RoboDK station: path.rdk

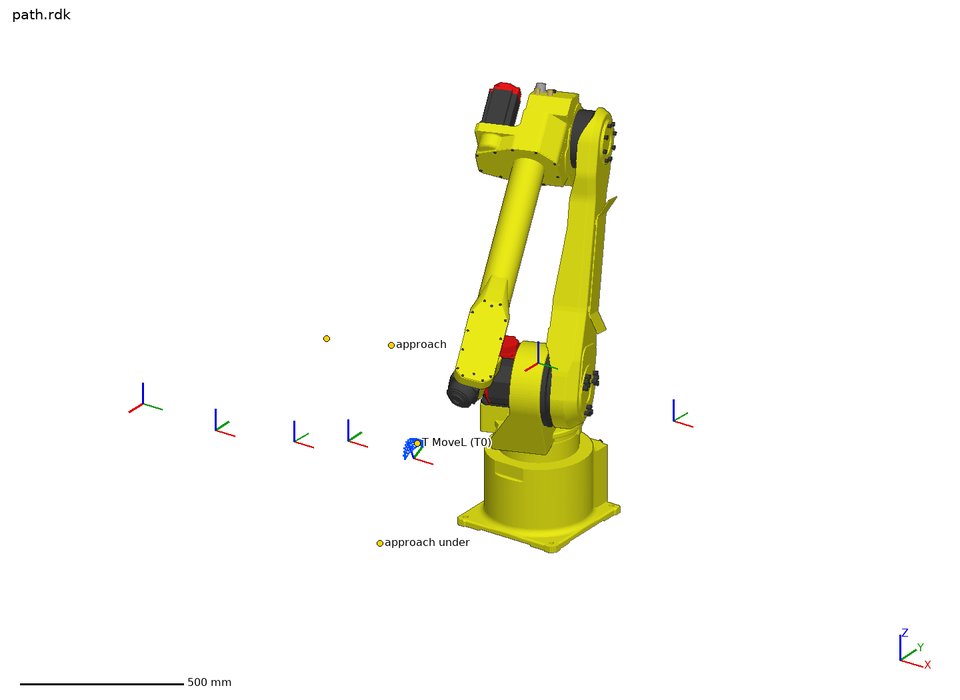
[picture v0: the station drawn from its stored meshes, robots at their saved joint values, targets as dots, program paths as lines]
Station path (saved by RoboDK 5.0.0). Poses are relative to the parent item; angles as X-Y-Z fixed-axis rotations.
  - frame data_frame at (0, 0, 0) mm
    - target approach (Cartesian target) at (94, 380, 204.2) mm, rotated rx -180 ry 0 rz 0 deg; joints [10.247, -49.52, -8.659, -50.211, 13.385, 139.433] of Fanuc ARC Mate 120iB/10L
    - target approach_vert (Cartesian target) at (0, 170, 284.2) mm, rotated rx -90 ry 0 rz 180 deg; joints [0, 2.156, 3.881, -180, 93.881, 90] of Fanuc ARC Mate 120iB/10L
    - target approach under (Cartesian target) at (94, 320, -445.8) mm; joints [3.897, 48.417, -53.03, 175.127, 126.871, 267.072] of Fanuc ARC Mate 120iB/10L
    - target approach_vert_180 (Cartesian target) at (0, 170, 284.2) mm, rotated rx -90 ry 0 rz 0 deg; joints [0, 2.156, 3.881, -180, 93.881, -90] of Fanuc ARC Mate 120iB/10L
    - frame data_frame_sphere at (270, 250, -80) mm, rotated rx 25 ry 0 rz 0 deg
      - object path at (0, 0, 0) mm, geometry from ible
      - target T MoveL (T0) (Cartesian target) at (-12.84, 46.05, 14.64) mm, rotated rx 112.92 ry -41.25 rz 0 deg; joints [16.302, 22.375, -63.434, -8.779, 128.992, 144.295] of Fanuc ARC Mate 120iB/10L
    - frame data_frame_zcyl at (-610, 450, -310) mm
    - frame data_frame_ycyl at (890, 750, 20) mm
    - frame data_frame_xcyl at (130, 100, 0) mm
    - frame data_frame_delta at (-1050, 690, -440) mm, rotated rx 0 ry 0 rz -90 deg
  - frame Fanuc ARC Mate 120iB/10L Base at (0, 1300, -250) mm, rotated rx 0 ry 0 rz -90 deg
    - robot Fanuc ARC Mate 120iB/10L: 6 axes, payload 10 kg, reach 1885 mm, repeatability 0.1 mm, weight 225 kg
        modified DH rows (alpha deg, a mm, theta deg, d mm): 0, 0, 0, 525; -90, 150, -90, 0; 0, 770, 0, 0; -90, 100, 0, 960; 90, 0, 0, 0; -90, 0, 0, 100
        base shift (0, 0, -525) mm
        joint limits [-170, -80, -170, -200, -140, -2160] to [170, 170, 250, 200, 140, 2160]; home [0, 0, 0, 0, 0, 0]; saved at [20.227, -18.261, -31.301, 104.445, -18.879, 20.92]
      - tool Tool 1, TCP at (0, 0, 300) mm, rotated rx 90 ry 0 rz 0 deg
      - tool Tool Normal, TCP at (0, 0, 200) mm
      - tool Tool 3, TCP at (0, 0, 300) mm, rotated rx -90 ry 0 rz 0 deg
      - tool Tool OD Orient, TCP at (0, 0, 300) mm, rotated rx 0 ry 90 rz -90 deg
      - tool Tool Sphere, TCP at (0, 0, 200) mm, rotated rx 0 ry 0 rz 45 deg
  - program AutoProgram (201 instructions, listed below)
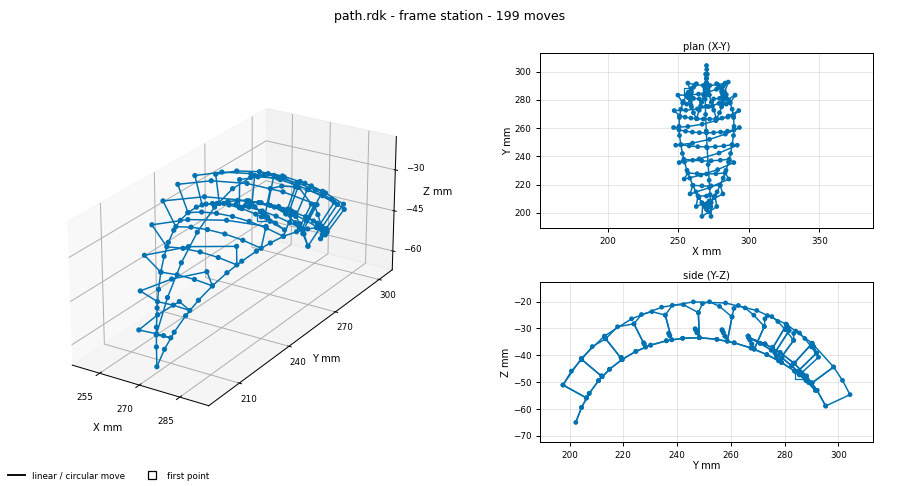
[picture p0: tool path of path.rdk in frame station, 199 of 199 moves have a stored position in this frame; points joined in program order, loops and branches not executed]

--- program AutoProgram (robot Fanuc ARC Mate 120iB/10L) ---
  Set Ref.: data_frame_sphere
  Set Tool: Tool Sphere
  *MoveL (T0) -> target T MoveL (T0)
  MoveL (T1) to (-11.94, 46.05, 15.38) mm, rotated rx 112.92 ry -37.81 rz 0 deg; joints [16.302, 22.375, -63.434, -8.779, 128.992, 144.295]
  MoveL (T2) to (-10.99, 46.05, 16.07) mm, rotated rx 112.92 ry -34.38 rz 0 deg; joints [16.302, 22.375, -63.434, -8.779, 128.992, 144.295]
  MoveL (T3) to (-13.19, 55.26, 19.28) mm, rotated rx 112.92 ry -34.38 rz 0 deg; joints [16.302, 22.375, -63.434, -8.779, 128.992, 144.295]
  MoveL (T4) to (-8.01, 55.26, 21.95) mm, rotated rx 112.92 ry -20.05 rz 0 deg; joints [16.302, 22.375, -63.434, -8.779, 128.992, 144.295]
  MoveL (T5) to (-2.33, 55.26, 23.25) mm, rotated rx 112.92 ry -5.73 rz 0 deg; joints [16.302, 22.375, -63.434, -8.779, 128.992, 144.295]
  MoveL (T6) to (-1.94, 46.05, 19.37) mm, rotated rx 112.92 ry -5.73 rz 0 deg; joints [16.302, 22.375, -63.434, -8.779, 128.992, 144.295]
  MoveL (T7) to (0, 46.05, 19.47) mm, rotated rx 112.92 ry 0 rz 0 deg; joints [16.302, 22.375, -63.434, -8.779, 128.992, 144.295]
  MoveL (T8) to (1.94, 46.05, 19.37) mm, rotated rx 112.92 ry 5.73 rz 0 deg; joints [16.302, 22.375, -63.434, -8.779, 128.992, 144.295]
  MoveL (T9) to (2.33, 55.26, 23.25) mm, rotated rx 112.92 ry 5.73 rz 0 deg; joints [16.302, 22.375, -63.434, -8.779, 128.992, 144.295]
  MoveL (T10) to (8.01, 55.26, 21.95) mm, rotated rx 112.92 ry 20.05 rz 0 deg; joints [16.302, 22.375, -63.434, -8.779, 128.992, 144.295]
  MoveL (T11) to (13.19, 55.26, 19.28) mm, rotated rx 112.92 ry 34.38 rz 0 deg; joints [16.302, 22.375, -63.434, -8.779, 128.992, 144.295]
  MoveL (T12) to (10.99, 46.05, 16.07) mm, rotated rx 112.92 ry 34.38 rz 0 deg; joints [16.302, 22.375, -63.434, -8.779, 128.992, 144.295]
  MoveL (T13) to (11.94, 46.05, 15.38) mm, rotated rx 112.92 ry 37.81 rz 0 deg; joints [16.302, 22.375, -63.434, -8.779, 128.992, 144.295]
  MoveL (T14) to (12.84, 46.05, 14.64) mm, rotated rx 112.92 ry 41.25 rz 0 deg; joints [16.302, 22.375, -63.434, -8.779, 128.992, 144.295]
  MoveL (T15) to (15.41, 55.26, 17.57) mm, rotated rx 112.92 ry 41.25 rz 0 deg; joints [16.302, 22.375, -63.434, -8.779, 128.992, 144.295]
  MoveL (T16) to (11.93, 54.45, 22.19) mm, rotated rx 114.83 ry 28.27 rz 0 deg; joints [16.302, 22.375, -63.434, -8.779, 128.992, 144.295]
  MoveL (T17) to (7.11, 53.58, 26.04) mm, rotated rx 116.74 ry 15.28 rz 0 deg; joints [16.302, 22.375, -63.434, -8.779, 128.992, 144.295]
  MoveL (T18) to (1.15, 52.66, 28.74) mm, rotated rx 118.65 ry 2.29 rz 0 deg; joints [16.302, 22.375, -63.434, -8.779, 128.992, 144.295]
  MoveL (T19) to (-5.66, 51.67, 29.97) mm, rotated rx 120.56 ry -10.7 rz 0 deg; joints [16.302, 22.375, -63.434, -8.779, 128.992, 144.295]
  MoveL (T20) to (-12.94, 50.62, 29.5) mm, rotated rx 122.47 ry -23.68 rz 0 deg; joints [16.302, 22.375, -63.434, -8.779, 128.992, 144.295]
  MoveL (T21) to (-20.23, 49.52, 27.17) mm, rotated rx 124.38 ry -36.67 rz 0 deg; joints [16.302, 22.375, -63.434, -8.779, 128.992, 144.295]
  MoveL (T22) to (-16.86, 41.27, 22.64) mm, rotated rx 124.38 ry -36.67 rz 0 deg; joints [16.302, 22.375, -63.434, -8.779, 128.992, 144.295]
  MoveL (T23) to (-14.03, 41.27, 24.5) mm, rotated rx 124.38 ry -29.79 rz 0 deg; joints [16.302, 22.375, -63.434, -8.779, 128.992, 144.295]
  MoveL (T24) to (-10.99, 41.27, 26) mm, rotated rx 124.38 ry -22.92 rz 0 deg; joints [16.302, 22.375, -63.434, -8.779, 128.992, 144.295]
  MoveL (T25) to (-13.19, 49.52, 31.2) mm, rotated rx 124.38 ry -22.92 rz 0 deg; joints [16.302, 22.375, -63.434, -8.779, 128.992, 144.295]
  MoveL (T26) to (-9.2, 49.52, 32.61) mm, rotated rx 124.38 ry -15.76 rz 0 deg; joints [16.302, 22.375, -63.434, -8.779, 128.992, 144.295]
  MoveL (T27) to (-5.06, 49.52, 33.5) mm, rotated rx 124.38 ry -8.59 rz 0 deg; joints [16.302, 22.375, -63.434, -8.779, 128.992, 144.295]
  MoveL (T28) to (-4.22, 41.27, 27.91) mm, rotated rx 124.38 ry -8.59 rz 0 deg; joints [16.302, 22.375, -63.434, -8.779, 128.992, 144.295]
  MoveL (T29) to (0, 41.27, 28.23) mm, rotated rx 124.38 ry 0 rz 0 deg; joints [16.302, 22.375, -63.434, -8.779, 128.992, 144.295]
  MoveL (T30) to (4.22, 41.27, 27.91) mm, rotated rx 124.38 ry 8.59 rz 0 deg; joints [16.302, 22.375, -63.434, -8.779, 128.992, 144.295]
  MoveL (T31) to (5.06, 49.52, 33.5) mm, rotated rx 124.38 ry 8.59 rz 0 deg; joints [16.302, 22.375, -63.434, -8.779, 128.992, 144.295]
  MoveL (T32) to (9.2, 49.52, 32.61) mm, rotated rx 124.38 ry 15.76 rz 0 deg; joints [16.302, 22.375, -63.434, -8.779, 128.992, 144.295]
  MoveL (T33) to (13.19, 49.52, 31.2) mm, rotated rx 124.38 ry 22.92 rz 0 deg; joints [16.302, 22.375, -63.434, -8.779, 128.992, 144.295]
  MoveL (T34) to (10.99, 41.27, 26) mm, rotated rx 124.38 ry 22.92 rz 0 deg; joints [16.302, 22.375, -63.434, -8.779, 128.992, 144.295]
  MoveL (T35) to (14.03, 41.27, 24.5) mm, rotated rx 124.38 ry 29.79 rz 0 deg; joints [16.302, 22.375, -63.434, -8.779, 128.992, 144.295]
  MoveL (T36) to (16.86, 41.27, 22.64) mm, rotated rx 124.38 ry 36.67 rz 0 deg; joints [16.302, 22.375, -63.434, -8.779, 128.992, 144.295]
  MoveL (T37) to (20.23, 49.52, 27.17) mm, rotated rx 124.38 ry 36.67 rz 0 deg; joints [16.302, 22.375, -63.434, -8.779, 128.992, 144.295]
  MoveL (T38) to (15.12, 48.36, 32.13) mm, rotated rx 126.29 ry 25.21 rz 0 deg; joints [16.302, 22.375, -63.434, -8.779, 128.992, 144.295]
  MoveL (T39) to (8.82, 47.15, 36.04) mm, rotated rx 128.2 ry 13.75 rz 0 deg; joints [16.302, 22.375, -63.434, -8.779, 128.992, 144.295]
  MoveL (T40) to (1.55, 45.89, 38.62) mm, rotated rx 130.11 ry 2.29 rz 0 deg; joints [16.302, 22.375, -63.434, -8.779, 128.992, 144.295]
  MoveL (T41) to (-6.4, 44.58, 39.65) mm, rotated rx 132.02 ry -9.17 rz 0 deg; joints [16.302, 22.375, -63.434, -8.779, 128.992, 144.295]
  MoveL (T42) to (-14.66, 43.21, 38.96) mm, rotated rx 133.93 ry -20.63 rz 0 deg; joints [16.302, 22.375, -63.434, -8.779, 128.992, 144.295]
  MoveL (T43) to (-22.86, 41.8, 36.47) mm, rotated rx 135.84 ry -32.09 rz 0 deg; joints [16.302, 22.375, -63.434, -8.779, 128.992, 144.295]
  MoveL (T44) to (-19.05, 34.84, 30.39) mm, rotated rx 135.84 ry -32.09 rz 0 deg; joints [16.302, 22.375, -63.434, -8.779, 128.992, 144.295]
  MoveL (T45) to (-15.13, 34.84, 32.52) mm, rotated rx 135.84 ry -24.96 rz 0 deg; joints [16.302, 22.375, -63.434, -8.779, 128.992, 144.295]
  MoveL (T46) to (-10.98, 34.84, 34.15) mm, rotated rx 135.84 ry -17.83 rz 0 deg; joints [16.302, 22.375, -63.434, -8.779, 128.992, 144.295]
  MoveL (T47) to (-6.66, 34.84, 35.24) mm, rotated rx 135.84 ry -10.7 rz 0 deg; joints [16.302, 22.375, -63.434, -8.779, 128.992, 144.295]
  MoveL (T48) to (-2.23, 34.84, 35.8) mm, rotated rx 135.84 ry -3.56 rz 0 deg; joints [16.302, 22.375, -63.434, -8.779, 128.992, 144.295]
  MoveL (T49) to (2.23, 34.84, 35.8) mm, rotated rx 135.84 ry 3.56 rz 0 deg; joints [16.302, 22.375, -63.434, -8.779, 128.992, 144.295]
  MoveL (T50) to (6.66, 34.84, 35.24) mm, rotated rx 135.84 ry 10.7 rz 0 deg; joints [16.302, 22.375, -63.434, -8.779, 128.992, 144.295]
  MoveL (T51) to (10.98, 34.84, 34.15) mm, rotated rx 135.84 ry 17.83 rz 0 deg; joints [16.302, 22.375, -63.434, -8.779, 128.992, 144.295]
  MoveL (T52) to (15.13, 34.84, 32.52) mm, rotated rx 135.84 ry 24.96 rz 0 deg; joints [16.302, 22.375, -63.434, -8.779, 128.992, 144.295]
  MoveL (T53) to (19.05, 34.84, 30.39) mm, rotated rx 135.84 ry 32.09 rz 0 deg; joints [16.302, 22.375, -63.434, -8.779, 128.992, 144.295]
  MoveL (T54) to (22.86, 41.8, 36.47) mm, rotated rx 135.84 ry 32.09 rz 0 deg; joints [16.302, 22.375, -63.434, -8.779, 128.992, 144.295]
  MoveL (T55) to (15.4, 40.05, 41.94) mm, rotated rx 138.13 ry 20.17 rz 0 deg; joints [16.302, 22.375, -63.434, -8.779, 128.992, 144.295]
  MoveL (T56) to (6.64, 38.23, 45.77) mm, rotated rx 140.42 ry 8.25 rz 0 deg; joints [16.302, 22.375, -63.434, -8.779, 128.992, 144.295]
  MoveL (T57) to (-3.05, 36.35, 47.64) mm, rotated rx 142.71 ry -3.67 rz 0 deg; joints [16.302, 22.375, -63.434, -8.779, 128.992, 144.295]
  MoveL (T58) to (-13.21, 34.41, 47.34) mm, rotated rx 145 ry -15.58 rz 0 deg; joints [16.302, 22.375, -63.434, -8.779, 128.992, 144.295]
  MoveL (T59) to (-23.31, 32.42, 44.78) mm, rotated rx 147.3 ry -27.5 rz 0 deg; joints [16.302, 22.375, -63.434, -8.779, 128.992, 144.295]
  MoveL (T60) to (-19.43, 27.02, 37.32) mm, rotated rx 147.3 ry -27.5 rz 0 deg; joints [16.302, 22.375, -63.434, -8.779, 128.992, 144.295]
  MoveL (T61) to (-14.82, 27.02, 39.38) mm, rotated rx 147.3 ry -20.63 rz 0 deg; joints [16.302, 22.375, -63.434, -8.779, 128.992, 144.295]
  MoveL (T62) to (-10, 27.02, 40.87) mm, rotated rx 147.3 ry -13.75 rz 0 deg; joints [16.302, 22.375, -63.434, -8.779, 128.992, 144.295]
  MoveL (T63) to (-5.04, 27.02, 41.77) mm, rotated rx 147.3 ry -6.88 rz 0 deg; joints [16.302, 22.375, -63.434, -8.779, 128.992, 144.295]
  MoveL (T64) to (0, 27.02, 42.07) mm, rotated rx 147.3 ry 0 rz 0 deg; joints [16.302, 22.375, -63.434, -8.779, 128.992, 144.295]
  MoveL (T65) to (5.04, 27.02, 41.77) mm, rotated rx 147.3 ry 6.88 rz 0 deg; joints [16.302, 22.375, -63.434, -8.779, 128.992, 144.295]
  MoveL (T66) to (10, 27.02, 40.87) mm, rotated rx 147.3 ry 13.75 rz 0 deg; joints [16.302, 22.375, -63.434, -8.779, 128.992, 144.295]
  MoveL (T67) to (14.82, 27.02, 39.38) mm, rotated rx 147.3 ry 20.63 rz 0 deg; joints [16.302, 22.375, -63.434, -8.779, 128.992, 144.295]
  MoveL (T68) to (19.43, 27.02, 37.32) mm, rotated rx 147.3 ry 27.5 rz 0 deg; joints [16.302, 22.375, -63.434, -8.779, 128.992, 144.295]
  MoveL (T69) to (23.31, 32.42, 44.78) mm, rotated rx 147.3 ry 27.5 rz 0 deg; joints [16.302, 22.375, -63.434, -8.779, 128.992, 144.295]
  MoveL (T70) to (13.38, 29.85, 50.3) mm, rotated rx 150.16 ry 14.9 rz 0 deg; joints [16.302, 22.375, -63.434, -8.779, 128.992, 144.295]
  MoveL (T71) to (2.14, 27.22, 53.43) mm, rotated rx 153.03 ry 2.29 rz 0 deg; joints [16.302, 22.375, -63.434, -8.779, 128.992, 144.295]
  MoveL (T72) to (-9.8, 24.51, 53.88) mm, rotated rx 155.89 ry -10.31 rz 0 deg; joints [16.302, 22.375, -63.434, -8.779, 128.992, 144.295]
  MoveL (T73) to (-21.78, 21.74, 51.51) mm, rotated rx 158.75 ry -22.92 rz 0 deg; joints [16.302, 22.375, -63.434, -8.779, 128.992, 144.295]
  MoveL (T74) to (-18.15, 18.12, 42.92) mm, rotated rx 158.75 ry -22.92 rz 0 deg; joints [16.302, 22.375, -63.434, -8.779, 128.992, 144.295]
  MoveL (T75) to (-12.28, 18.12, 44.95) mm, rotated rx 158.75 ry -15.28 rz 0 deg; joints [16.302, 22.375, -63.434, -8.779, 128.992, 144.295]
  MoveL (T76) to (-6.2, 18.12, 46.19) mm, rotated rx 158.75 ry -7.64 rz 0 deg; joints [16.302, 22.375, -63.434, -8.779, 128.992, 144.295]
  MoveL (T77) to (0, 18.12, 46.6) mm, rotated rx 158.75 ry 0 rz 0 deg; joints [16.302, 22.375, -63.434, -8.779, 128.992, 144.295]
  MoveL (T78) to (6.2, 18.12, 46.19) mm, rotated rx 158.75 ry 7.64 rz 0 deg; joints [16.302, 22.375, -63.434, -8.779, 128.992, 144.295]
  MoveL (T79) to (12.28, 18.12, 44.95) mm, rotated rx 158.75 ry 15.28 rz 0 deg; joints [16.302, 22.375, -63.434, -8.779, 128.992, 144.295]
  MoveL (T80) to (18.15, 18.12, 42.92) mm, rotated rx 158.75 ry 22.92 rz 0 deg; joints [16.302, 22.375, -63.434, -8.779, 128.992, 144.295]
  MoveL (T81) to (21.78, 21.74, 51.51) mm, rotated rx 158.75 ry 22.92 rz 0 deg; joints [16.302, 22.375, -63.434, -8.779, 128.992, 144.295]
  MoveL (T82) to (8.87, 17.97, 56.55) mm, rotated rx 162.57 ry 8.91 rz 0 deg; joints [16.302, 22.375, -63.434, -8.779, 128.992, 144.295]
  MoveL (T83) to (-5.18, 14.11, 58.09) mm, rotated rx 166.39 ry -5.09 rz 0 deg; joints [16.302, 22.375, -63.434, -8.779, 128.992, 144.295]
  MoveL (T84) to (-19.35, 10.2, 55.87) mm, rotated rx 170.21 ry -19.1 rz 0 deg; joints [16.302, 22.375, -63.434, -8.779, 128.992, 144.295]
  MoveL (T85) to (-16.12, 8.5, 46.56) mm, rotated rx 170.21 ry -19.1 rz 0 deg; joints [16.302, 22.375, -63.434, -8.779, 128.992, 144.295]
  MoveL (T86) to (-9.79, 8.5, 48.29) mm, rotated rx 170.21 ry -11.46 rz 0 deg; joints [16.302, 22.375, -63.434, -8.779, 128.992, 144.295]
  MoveL (T87) to (-3.28, 8.5, 49.16) mm, rotated rx 170.21 ry -3.82 rz 0 deg; joints [16.302, 22.375, -63.434, -8.779, 128.992, 144.295]
  MoveL (T88) to (3.28, 8.5, 49.16) mm, rotated rx 170.21 ry 3.82 rz 0 deg; joints [16.302, 22.375, -63.434, -8.779, 128.992, 144.295]
  MoveL (T89) to (9.79, 8.5, 48.29) mm, rotated rx 170.21 ry 11.46 rz 0 deg; joints [16.302, 22.375, -63.434, -8.779, 128.992, 144.295]
  MoveL (T90) to (16.12, 8.5, 46.56) mm, rotated rx 170.21 ry 19.1 rz 0 deg; joints [16.302, 22.375, -63.434, -8.779, 128.992, 144.295]
  MoveL (T91) to (19.35, 10.2, 55.87) mm, rotated rx 170.21 ry 19.1 rz 0 deg; joints [16.302, 22.375, -63.434, -8.779, 128.992, 144.295]
  MoveL (T92) to (7.93, 6.24, 59.15) mm, rotated rx 174.03 ry 7.64 rz 0 deg; joints [16.302, 22.375, -63.434, -8.779, 128.992, 144.295]
  MoveL (T93) to (-3.99, 2.25, 59.83) mm, rotated rx 177.85 ry -3.82 rz 0 deg; joints [16.302, 22.375, -63.434, -8.779, 128.992, 144.295]
  MoveL (T94) to (-15.8, -1.75, 57.85) mm, rotated rx -178.33 ry -15.28 rz 0 deg; joints [16.302, 22.375, -63.434, -8.779, 128.992, 144.295]
  MoveL (T95) to (-13.17, -1.46, 48.21) mm, rotated rx -178.33 ry -15.28 rz 0 deg; joints [16.302, 22.375, -63.434, -8.779, 128.992, 144.295]
  MoveL (T96) to (-6.64, -1.46, 49.53) mm, rotated rx -178.33 ry -7.64 rz 0 deg; joints [16.302, 22.375, -63.434, -8.779, 128.992, 144.295]
  MoveL (T97) to (0, -1.46, 49.98) mm, rotated rx -178.33 ry 0 rz 0 deg; joints [16.302, 22.375, -63.434, -8.779, 128.992, 144.295]
  MoveL (T98) to (6.64, -1.46, 49.53) mm, rotated rx -178.33 ry 7.64 rz 0 deg; joints [16.302, 22.375, -63.434, -8.779, 128.992, 144.295]
  MoveL (T99) to (13.17, -1.46, 48.21) mm, rotated rx -178.33 ry 15.28 rz 0 deg; joints [16.302, 22.375, -63.434, -8.779, 128.992, 144.295]
  MoveL (T100) to (15.8, -1.75, 57.85) mm, rotated rx -178.33 ry 15.28 rz 0 deg; joints [16.302, 22.375, -63.434, -8.779, 128.992, 144.295]
  MoveL (T101) to (1.98, -7.73, 59.47) mm, rotated rx -172.6 ry 1.91 rz 0 deg; joints [16.302, 22.375, -63.434, -8.779, 128.992, 144.295]
  MoveL (T102) to (-11.61, -13.63, 57.27) mm, rotated rx -166.87 ry -11.46 rz 0 deg; joints [16.302, 22.375, -63.434, -8.779, 128.992, 144.295]
  MoveL (T103) to (-9.67, -11.36, 47.72) mm, rotated rx -166.87 ry -11.46 rz 0 deg; joints [16.302, 22.375, -63.434, -8.779, 128.992, 144.295]
  MoveL (T104) to (-3.24, -11.36, 48.58) mm, rotated rx -166.87 ry -3.82 rz 0 deg; joints [16.302, 22.375, -63.434, -8.779, 128.992, 144.295]
  MoveL (T105) to (3.24, -11.36, 48.58) mm, rotated rx -166.87 ry 3.82 rz 0 deg; joints [16.302, 22.375, -63.434, -8.779, 128.992, 144.295]
  MoveL (T106) to (9.67, -11.36, 47.72) mm, rotated rx -166.87 ry 11.46 rz 0 deg; joints [16.302, 22.375, -63.434, -8.779, 128.992, 144.295]
  MoveL (T107) to (11.61, -13.63, 57.27) mm, rotated rx -166.87 ry 11.46 rz 0 deg; joints [16.302, 22.375, -63.434, -8.779, 128.992, 144.295]
  MoveL (T108) to (1.89, -19.4, 56.75) mm, rotated rx -161.14 ry 1.91 rz 0 deg; joints [16.302, 22.375, -63.434, -8.779, 128.992, 144.295]
  MoveL (T109) to (-7.25, -24.97, 54.07) mm, rotated rx -155.41 ry -7.64 rz 0 deg; joints [16.302, 22.375, -63.434, -8.779, 128.992, 144.295]
  MoveL (T110) to (-6.04, -20.81, 45.06) mm, rotated rx -155.41 ry -7.64 rz 0 deg; joints [16.302, 22.375, -63.434, -8.779, 128.992, 144.295]
  MoveL (T111) to (0, -20.81, 45.47) mm, rotated rx -155.41 ry 0 rz 0 deg; joints [16.302, 22.375, -63.434, -8.779, 128.992, 144.295]
  MoveL (T112) to (6.04, -20.81, 45.06) mm, rotated rx -155.41 ry 7.64 rz 0 deg; joints [16.302, 22.375, -63.434, -8.779, 128.992, 144.295]
  MoveL (T113) to (7.25, -24.97, 54.07) mm, rotated rx -155.41 ry 7.64 rz 0 deg; joints [16.302, 22.375, -63.434, -8.779, 128.992, 144.295]
  MoveL (T114) to (1.73, -30.29, 51.76) mm, rotated rx -149.68 ry 1.91 rz 0 deg; joints [16.302, 22.375, -63.434, -8.779, 128.992, 144.295]
  MoveL (T115) to (-3.23, -35.31, 48.4) mm, rotated rx -143.95 ry -3.82 rz 0 deg; joints [16.302, 22.375, -63.434, -8.779, 128.992, 144.295]
  MoveL (T116) to (-2.69, -29.43, 40.34) mm, rotated rx -143.95 ry -3.82 rz 0 deg; joints [16.302, 22.375, -63.434, -8.779, 128.992, 144.295]
  MoveL (T117) to (0, -29.43, 40.42) mm, rotated rx -143.95 ry 0 rz 0 deg; joints [16.302, 22.375, -63.434, -8.779, 128.992, 144.295]
  MoveL (T118) to (2.69, -29.43, 40.34) mm, rotated rx -143.95 ry 3.82 rz 0 deg; joints [16.302, 22.375, -63.434, -8.779, 128.992, 144.295]
  MoveL (T119) to (3.23, -35.31, 48.4) mm, rotated rx -143.95 ry 3.82 rz 0 deg; joints [16.302, 22.375, -63.434, -8.779, 128.992, 144.295]
  MoveL (T120) to (3, -24.97, 54.48) mm, rotated rx -155.41 ry 3.15 rz 0 deg; joints [16.302, 22.375, -63.434, -8.779, 128.992, 144.295]
  MoveL (T121) to (2.53, -13.63, 58.38) mm, rotated rx -166.87 ry 2.48 rz 0 deg; joints [16.302, 22.375, -63.434, -8.779, 128.992, 144.295]
  MoveL (T122) to (1.9, -1.75, 59.94) mm, rotated rx -178.33 ry 1.81 rz 0 deg; joints [16.302, 22.375, -63.434, -8.779, 128.992, 144.295]
  MoveL (T123) to (1.18, 10.2, 59.12) mm, rotated rx 170.21 ry 1.15 rz 0 deg; joints [16.302, 22.375, -63.434, -8.779, 128.992, 144.295]
  MoveL (T124) to (0.47, 21.74, 55.92) mm, rotated rx 158.75 ry 0.48 rz 0 deg; joints [16.302, 22.375, -63.434, -8.779, 128.992, 144.295]
  MoveL (T125) to (-0.17, 32.42, 50.49) mm, rotated rx 147.3 ry -0.19 rz 0 deg; joints [16.302, 22.375, -63.434, -8.779, 128.992, 144.295]
  MoveL (T126) to (-0.65, 41.8, 43.04) mm, rotated rx 135.84 ry -0.86 rz 0 deg; joints [16.302, 22.375, -63.434, -8.779, 128.992, 144.295]
  MoveL (T127) to (-0.9, 49.52, 33.87) mm, rotated rx 124.38 ry -1.53 rz 0 deg; joints [16.302, 22.375, -63.434, -8.779, 128.992, 144.295]
  MoveL (T128) to (-0.9, 55.26, 23.35) mm, rotated rx 112.92 ry -2.2 rz 0 deg; joints [16.302, 22.375, -63.434, -8.779, 128.992, 144.295]
  MoveL (T129) to (-0.59, 58.8, 11.9) mm, rotated rx 101.46 ry -2.87 rz 0 deg; joints [16.302, 22.375, -63.434, -8.779, 128.992, 144.295]
  MoveL (T130) to (-0.5, 49, 9.92) mm, rotated rx 101.46 ry -2.87 rz 0 deg; joints [16.302, 22.375, -63.434, -8.779, 128.992, 144.295]
  MoveL (T131) to (0, 49, 9.93) mm, rotated rx 101.46 ry 0 rz 0 deg; joints [16.302, 22.375, -63.434, -8.779, 128.992, 144.295]
  MoveL (T132) to (0.5, 49, 9.92) mm, rotated rx 101.46 ry 2.87 rz 0 deg; joints [16.302, 22.375, -63.434, -8.779, 128.992, 144.295]
  MoveL (T133) to (0.59, 58.8, 11.9) mm, rotated rx 101.46 ry 2.87 rz 0 deg; joints [16.302, 22.375, -63.434, -8.779, 128.992, 144.295]
  MoveL (T134) to (0.15, 59.7, 5.99) mm, rotated rx 95.73 ry 1.43 rz 0 deg; joints [16.302, 22.375, -63.434, -8.779, 128.992, 144.295]
  MoveL (T135) to (0, 60, 0) mm, rotated rx 90 ry 0 rz 0 deg; joints [16.302, 22.375, -63.434, -8.779, 128.992, 144.295]
  MoveL (T136) to (0, 50, 0) mm, rotated rx 90 ry 0 rz 0 deg; joints [16.302, 22.375, -63.434, -8.779, 128.992, 144.295]
  MoveL (T137) to (0.22, 49.56, 6.64) mm, rotated rx 97.64 ry 1.91 rz 0 deg; joints [16.302, 22.375, -63.434, -8.779, 128.992, 144.295]
  MoveL (T138) to (0.88, 48.23, 13.15) mm, rotated rx 105.28 ry 3.82 rz 0 deg; joints [16.302, 22.375, -63.434, -8.779, 128.992, 144.295]
  MoveL (T139) to (1.94, 46.05, 19.37) mm, rotated rx 112.92 ry 5.73 rz 0 deg; joints [16.302, 22.375, -63.434, -8.779, 128.992, 144.295]
  MoveL (T140) to (3.38, 43.06, 25.2) mm, rotated rx 120.56 ry 7.64 rz 0 deg; joints [16.302, 22.375, -63.434, -8.779, 128.992, 144.295]
  MoveL (T141) to (5.13, 39.29, 30.49) mm, rotated rx 128.2 ry 9.55 rz 0 deg; joints [16.302, 22.375, -63.434, -8.779, 128.992, 144.295]
  MoveL (T142) to (7.13, 34.84, 35.15) mm, rotated rx 135.84 ry 11.46 rz 0 deg; joints [16.302, 22.375, -63.434, -8.779, 128.992, 144.295]
  MoveL (T143) to (9.23, 37.78, 31.43) mm, rotated rx 130.93 ry 16.37 rz 0 deg; joints [16.302, 22.375, -63.434, -8.779, 128.992, 144.295]
  MoveL (T144) to (10.67, 40.44, 27.39) mm, rotated rx 126.02 ry 21.28 rz 0 deg; joints [16.302, 22.375, -63.434, -8.779, 128.992, 144.295]
  MoveL (T145) to (11.4, 42.81, 23.18) mm, rotated rx 121.1 ry 26.19 rz 0 deg; joints [16.302, 22.375, -63.434, -8.779, 128.992, 144.295]
  MoveL (T146) to (11.4, 44.87, 18.9) mm, rotated rx 116.19 ry 31.1 rz 0 deg; joints [16.302, 22.375, -63.434, -8.779, 128.992, 144.295]
  MoveL (T147) to (10.67, 46.59, 14.68) mm, rotated rx 111.28 ry 36.02 rz 0 deg; joints [16.302, 22.375, -63.434, -8.779, 128.992, 144.295]
  MoveL (T148) to (9.23, 47.97, 10.65) mm, rotated rx 106.37 ry 40.93 rz 0 deg; joints [16.302, 22.375, -63.434, -8.779, 128.992, 144.295]
  MoveL (T149) to (7.13, 49, 6.92) mm, rotated rx 101.46 ry 45.84 rz 0 deg; joints [16.302, 22.375, -63.434, -8.779, 128.992, 144.295]
  MoveL (T150) to (10.88, 47.38, 11.68) mm, rotated rx 108.62 ry 42.97 rz 0 deg; joints [16.302, 22.375, -63.434, -8.779, 128.992, 144.295]
  MoveL (T151) to (14.01, 45.02, 16.63) mm, rotated rx 115.78 ry 40.11 rz 0 deg; joints [16.302, 22.375, -63.434, -8.779, 128.992, 144.295]
  MoveL (T152) to (16.46, 41.96, 21.65) mm, rotated rx 122.94 ry 37.24 rz 0 deg; joints [16.302, 22.375, -63.434, -8.779, 128.992, 144.295]
  MoveL (T153) to (18.19, 38.24, 26.59) mm, rotated rx 130.11 ry 34.38 rz 0 deg; joints [16.302, 22.375, -63.434, -8.779, 128.992, 144.295]
  MoveL (T154) to (19.2, 33.93, 31.31) mm, rotated rx 137.27 ry 31.51 rz 0 deg; joints [16.302, 22.375, -63.434, -8.779, 128.992, 144.295]
  MoveL (T155) to (19.5, 29.08, 35.69) mm, rotated rx 144.43 ry 28.65 rz 0 deg; joints [16.302, 22.375, -63.434, -8.779, 128.992, 144.295]
  MoveL (T156) to (19.13, 23.79, 39.6) mm, rotated rx 151.59 ry 25.78 rz 0 deg; joints [16.302, 22.375, -63.434, -8.779, 128.992, 144.295]
  MoveL (T157) to (18.15, 18.12, 42.92) mm, rotated rx 158.75 ry 22.92 rz 0 deg; joints [16.302, 22.375, -63.434, -8.779, 128.992, 144.295]
  MoveL (T158) to (17.06, 12.41, 45.33) mm, rotated rx 165.63 ry 20.63 rz 0 deg; joints [16.302, 22.375, -63.434, -8.779, 128.992, 144.295]
  MoveL (T159) to (15.59, 6.52, 47.06) mm, rotated rx 172.51 ry 18.34 rz 0 deg; joints [16.302, 22.375, -63.434, -8.779, 128.992, 144.295]
  MoveL (T160) to (13.82, 0.54, 48.05) mm, rotated rx 179.38 ry 16.04 rz 0 deg; joints [16.302, 22.375, -63.434, -8.779, 128.992, 144.295]
  MoveL (T161) to (11.81, -5.45, 48.28) mm, rotated rx -173.74 ry 13.75 rz 0 deg; joints [16.302, 22.375, -63.434, -8.779, 128.992, 144.295]
  MoveL (T162) to (9.67, -11.36, 47.72) mm, rotated rx -166.87 ry 11.46 rz 0 deg; joints [16.302, 22.375, -63.434, -8.779, 128.992, 144.295]
  MoveL (T163) to (7.49, -17.11, 46.38) mm, rotated rx -159.99 ry 9.17 rz 0 deg; joints [16.302, 22.375, -63.434, -8.779, 128.992, 144.295]
  MoveL (T164) to (5.34, -22.61, 44.28) mm, rotated rx -153.12 ry 6.88 rz 0 deg; joints [16.302, 22.375, -63.434, -8.779, 128.992, 144.295]
  MoveL (T165) to (3.32, -27.79, 41.44) mm, rotated rx -146.24 ry 4.58 rz 0 deg; joints [16.302, 22.375, -63.434, -8.779, 128.992, 144.295]
  MoveL (T166) to (1.52, -32.56, 37.91) mm, rotated rx -139.37 ry 2.29 rz 0 deg; joints [16.302, 22.375, -63.434, -8.779, 128.992, 144.295]
  MoveL (T167) to (0, -36.87, 33.77) mm, rotated rx -132.49 ry 0 rz 0 deg; joints [16.302, 22.375, -63.434, -8.779, 128.992, 144.295]
  MoveL (T168) to (-1.52, -32.56, 37.91) mm, rotated rx -139.37 ry -2.29 rz 0 deg; joints [16.302, 22.375, -63.434, -8.779, 128.992, 144.295]
  MoveL (T169) to (-3.32, -27.79, 41.44) mm, rotated rx -146.24 ry -4.58 rz 0 deg; joints [16.302, 22.375, -63.434, -8.779, 128.992, 144.295]
  MoveL (T170) to (-5.34, -22.61, 44.28) mm, rotated rx -153.12 ry -6.88 rz 0 deg; joints [16.302, 22.375, -63.434, -8.779, 128.992, 144.295]
  MoveL (T171) to (-7.49, -17.11, 46.38) mm, rotated rx -159.99 ry -9.17 rz 0 deg; joints [16.302, 22.375, -63.434, -8.779, 128.992, 144.295]
  MoveL (T172) to (-9.67, -11.36, 47.72) mm, rotated rx -166.87 ry -11.46 rz 0 deg; joints [16.302, 22.375, -63.434, -8.779, 128.992, 144.295]
  MoveL (T173) to (-11.81, -5.45, 48.28) mm, rotated rx -173.74 ry -13.75 rz 0 deg; joints [16.302, 22.375, -63.434, -8.779, 128.992, 144.295]
  MoveL (T174) to (-13.82, 0.54, 48.05) mm, rotated rx 179.38 ry -16.04 rz 0 deg; joints [16.302, 22.375, -63.434, -8.779, 128.992, 144.295]
  MoveL (T175) to (-15.59, 6.52, 47.06) mm, rotated rx 172.51 ry -18.34 rz 0 deg; joints [16.302, 22.375, -63.434, -8.779, 128.992, 144.295]
  MoveL (T176) to (-17.06, 12.41, 45.33) mm, rotated rx 165.63 ry -20.63 rz 0 deg; joints [16.302, 22.375, -63.434, -8.779, 128.992, 144.295]
  MoveL (T177) to (-18.15, 18.12, 42.92) mm, rotated rx 158.75 ry -22.92 rz 0 deg; joints [16.302, 22.375, -63.434, -8.779, 128.992, 144.295]
  MoveL (T178) to (-19.13, 23.79, 39.6) mm, rotated rx 151.59 ry -25.78 rz 0 deg; joints [16.302, 22.375, -63.434, -8.779, 128.992, 144.295]
  MoveL (T179) to (-19.5, 29.08, 35.69) mm, rotated rx 144.43 ry -28.65 rz 0 deg; joints [16.302, 22.375, -63.434, -8.779, 128.992, 144.295]
  MoveL (T180) to (-19.2, 33.93, 31.31) mm, rotated rx 137.27 ry -31.51 rz 0 deg; joints [16.302, 22.375, -63.434, -8.779, 128.992, 144.295]
  MoveL (T181) to (-18.19, 38.24, 26.59) mm, rotated rx 130.11 ry -34.38 rz 0 deg; joints [16.302, 22.375, -63.434, -8.779, 128.992, 144.295]
  MoveL (T182) to (-16.46, 41.96, 21.65) mm, rotated rx 122.94 ry -37.24 rz 0 deg; joints [16.302, 22.375, -63.434, -8.779, 128.992, 144.295]
  MoveL (T183) to (-14.01, 45.02, 16.63) mm, rotated rx 115.78 ry -40.11 rz 0 deg; joints [16.302, 22.375, -63.434, -8.779, 128.992, 144.295]
  MoveL (T184) to (-10.88, 47.38, 11.68) mm, rotated rx 108.62 ry -42.97 rz 0 deg; joints [16.302, 22.375, -63.434, -8.779, 128.992, 144.295]
  MoveL (T185) to (-7.13, 49, 6.92) mm, rotated rx 101.46 ry -45.84 rz 0 deg; joints [16.302, 22.375, -63.434, -8.779, 128.992, 144.295]
  MoveL (T186) to (-9.23, 47.97, 10.65) mm, rotated rx 106.37 ry -40.93 rz 0 deg; joints [16.302, 22.375, -63.434, -8.779, 128.992, 144.295]
  MoveL (T187) to (-10.67, 46.59, 14.68) mm, rotated rx 111.28 ry -36.02 rz 0 deg; joints [16.302, 22.375, -63.434, -8.779, 128.992, 144.295]
  MoveL (T188) to (-11.4, 44.87, 18.9) mm, rotated rx 116.19 ry -31.1 rz 0 deg; joints [16.302, 22.375, -63.434, -8.779, 128.992, 144.295]
  MoveL (T189) to (-11.4, 42.81, 23.18) mm, rotated rx 121.1 ry -26.19 rz 0 deg; joints [16.302, 22.375, -63.434, -8.779, 128.992, 144.295]
  MoveL (T190) to (-10.67, 40.44, 27.39) mm, rotated rx 126.02 ry -21.28 rz 0 deg; joints [16.302, 22.375, -63.434, -8.779, 128.992, 144.295]
  MoveL (T191) to (-9.23, 37.78, 31.43) mm, rotated rx 130.93 ry -16.37 rz 0 deg; joints [16.302, 22.375, -63.434, -8.779, 128.992, 144.295]
  MoveL (T192) to (-7.13, 34.84, 35.15) mm, rotated rx 135.84 ry -11.46 rz 0 deg; joints [16.302, 22.375, -63.434, -8.779, 128.992, 144.295]
  MoveL (T193) to (-5.13, 39.29, 30.49) mm, rotated rx 128.2 ry -9.55 rz 0 deg; joints [16.302, 22.375, -63.434, -8.779, 128.992, 144.295]
  MoveL (T194) to (-3.38, 43.06, 25.2) mm, rotated rx 120.56 ry -7.64 rz 0 deg; joints [16.302, 22.375, -63.434, -8.779, 128.992, 144.295]
  MoveL (T195) to (-1.94, 46.05, 19.37) mm, rotated rx 112.92 ry -5.73 rz 0 deg; joints [16.302, 22.375, -63.434, -8.779, 128.992, 144.295]
  MoveL (T196) to (-0.88, 48.23, 13.15) mm, rotated rx 105.28 ry -3.82 rz 0 deg; joints [16.302, 22.375, -63.434, -8.779, 128.992, 144.295]
  MoveL (T197) to (-0.22, 49.56, 6.64) mm, rotated rx 97.64 ry -1.91 rz 0 deg; joints [16.302, 22.375, -63.434, -8.779, 128.992, 144.295]
  MoveL (T198) to (0, 50, 0) mm, rotated rx 90 ry 0 rz 0 deg; joints [16.302, 22.375, -63.434, -8.779, 128.992, 144.295]
